// TIA Portal V17 export
// export: Created 2023-04-11T09:33:27.8341102Z, ExportSetting WithDefaults, DisplayName Totally Integrated Automation Portal, DisplayVersion V17 Update 3, DisplayName TIA Portal Openness, DisplayVersion V17 Update 3, DisplayName TIA Portal Version Control Interface, DisplayVersion V17, DisplayName SINAMICS Startdrive Advanced, DisplayVersion V17 Update2, DisplayName SINAMICS Startdrive G130, G150, S120, S150, SINAMICS MV, S210, DisplayVersion V17 Update2, DisplayName SINAMICS Startdrive G110M, G120, G120C, G120D, G120P, G115D, DisplayVersion V17 Update2, DisplayName STEP 7 Professional, DisplayVersion V17 Update 3, DisplayName STEP 7 Safety, DisplayVersion V17, DisplayName WinCC UA Professional, DisplayVersion V17 Update 3
FUNCTION_BLOCK "FB_screenChangeControl"   // FB25, LAD
{ S7_Optimized_Access := 'TRUE' }
VERSION : 0.1
// stored: AutoNumber true, IsIECCheckEnabled false, IsRetainMemResEnabled false, MemoryReserve 100, SetENOAutomatically false, UDAEnableTagReadback false
   VAR_INPUT
      actualScreen : Int;
   END_VAR
   VAR_OUTPUT
      errorScrSwitch : Bool;
   END_VAR
   VAR_IN_OUT
      requestScreen_io : Int;
      changeEvent_io : SInt;
   END_VAR
   VAR
      edge : Array[0..1] of Bool;
      IEC_Timer_0_Instance { S7_SetPoint := 'True'} : TON_TIME;
      actualScreenBuffer : Int;
   END_VAR
   VAR_TEMP   // added for the SCL form of the ladder/FBD networks
      _w1 : Bool;
      _w2 : Bool;
      _w3 : Bool;
   END_VAR
BEGIN

REGION Network 1
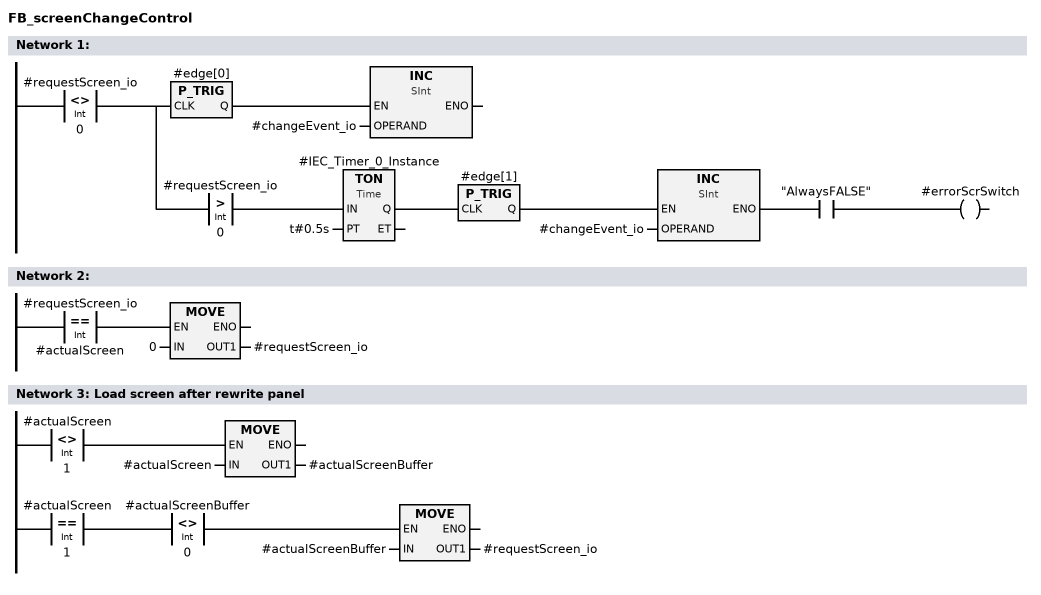
   RUNG wire#powerrail
      { S7_Templates := "SrcType := Int" } NE_Contact(in1 := #requestScreen_io, in2 := 0)
      wire#w1
      P_Trig( #edge[0] )
      { S7_Templates := "DestType := SInt" } Inc( #changeEvent_io )
   END_RUNG
   RUNG wire#w1
      { S7_Templates := "SrcType := Int" } GT_Contact(in1 := #requestScreen_io, in2 := 0)
      { S7_Templates := "time_type := Time" } #IEC_Timer_0_Instance.TON(pt := t#0.5s, et =>)
      P_Trig( #edge[1] )
      { S7_Templates := "DestType := SInt" } Inc( #changeEvent_io )
      Contact( "AlwaysFALSE" )
      Coil( #errorScrSwitch )
   END_RUNG
   // the same network as SCL:
   #_w1 := #requestScreen_io <> 0;
   #_w2 := #_w1 AND NOT #edge[0];   // rising edge
   #edge[0] := #_w1;
   IF #_w2 THEN #changeEvent_io := #changeEvent_io + 1; END_IF;
   #IEC_Timer_0_Instance(IN := #_w1 AND (#requestScreen_io > 0), PT := t#0.5s);   // TON
   #_w3 := #IEC_Timer_0_Instance.Q AND NOT #edge[1];   // rising edge
   #edge[1] := #IEC_Timer_0_Instance.Q;
   IF #_w3 THEN #changeEvent_io := #changeEvent_io + 1; END_IF;
   #errorScrSwitch := #_w3 AND "AlwaysFALSE";
END_REGION

REGION Network 2
   RUNG wire#powerrail
      { S7_Templates := "SrcType := Int" } EQ_Contact(in1 := #requestScreen_io, in2 := #actualScreen)
      Move(in := 0, out1 => #requestScreen_io)
   END_RUNG
   // the same network as SCL:
   IF #requestScreen_io = #actualScreen THEN #requestScreen_io := 0; END_IF;
END_REGION

REGION Network 3: Load screen after rewrite panel
   RUNG wire#powerrail
      { S7_Templates := "SrcType := Int" } NE_Contact(in1 := #actualScreen, in2 := 1)
      Move(in := #actualScreen, out1 => #actualScreenBuffer)
   END_RUNG
   RUNG wire#powerrail
      { S7_Templates := "SrcType := Int" } EQ_Contact(in1 := #actualScreen, in2 := 1)
      { S7_Templates := "SrcType := Int" } NE_Contact(in1 := #actualScreenBuffer, in2 := 0)
      Move(in := #actualScreenBuffer, out1 => #requestScreen_io)
   END_RUNG
   // the same network as SCL:
   IF #actualScreen <> 1 THEN #actualScreenBuffer := #actualScreen; END_IF;
   IF (#actualScreen = 1) AND (#actualScreenBuffer <> 0) THEN
       #requestScreen_io := #actualScreenBuffer;
   END_IF;
END_REGION
END_FUNCTION_BLOCK
